(* CODESYS project filling_station_1.ecp

Project tree, tasks and I/O mapping:
  GenericDummyMasterDevice : Generic Master, WAGO, order no. None, version 1.0.0.0
  PFC200_CS_2ETH_RS : 750-8202 PFC200 2ETH RS, WAGO, order no. 0750-8202, version 1.4.1.22
    application Application
      libraries: 
      task PLC_Task (cyclic, interval t#10ms, priority 14) calls PLC_PRG
      program PLC_PRG [ST]
    DeviceAdapter
    Kbus : Kbus, WAGO, version 1.3.0.0
        unmapped channels: K-BUS diagnostics
      _4_AI_0_10V_DC_s_e : 0750-0459, WAGO, order no. 0750-0459, version 0.0.0.11
          settings: K-BUS Module slot index = 2
          unmapped channels: _IW 1, _IW 2, _IW 3, _IW 4
        DeviceAdapter
      _2_AI_4_20mA_Diff_Measurement_Input : 0750-0492, WAGO, order no. 0750-0492, version 0.0.0.7
          settings: K-BUS Module slot index = 3
          unmapped channels: _IW 1, _IW 2
        DeviceAdapter
      _8_DO_Generic : 075x-8DO, WAGO, order no. 075x-8DO, version 0.0.0.11
          settings: K-BUS Module slot index = 1
          output output1 : BOOL  // _OUT._OUT
          output output2 : BOOL  // _OUT._OUT
          unmapped channels: _OUT
        DeviceAdapter
    MODBUS
      MODBUS : MODBUS, WAGO, order no. n/a, version 1.1.1.13
    Serial
      COM1 : COM1, WAGO, version 0.0.0.19
  Library Information/
    function GetLibVersion [ST]
    function GetLibVersionNumber [ST]
    function IsLibReleased [ST]
  Project Information/
    function GetTextProperty [ST]
    function GetTextProperty2 [ST]
    function GetNumberProperty [ST]
    function GetBooleanProperty [ST]
    function GetVersionProperty [ST]
    function GetCompany [ST]
    function GetTitle [ST]
    function GetVersion [ST]
*)

// PFC200_CS_2ETH_RS/Application/PLC_PRG
PROGRAM PLC_PRG
VAR
	Controller_OP_reversed: INT;
	vrValvePosition: INT;
	Water_Valve_Open: BOOL;
	Water_Valve_Close: BOOL;
	set: INT;
END_VAR

output1:=TRUE;
output2:=TRUE;

END_PROGRAM

// Library Information/GetLibVersion
// This function has been automatically generated from the project information.
FUNCTION GetLibVersion : VERSION
VAR_INPUT
	
END_VAR

GetLibVersion.uiMajor := 0;
GetLibVersion.uiMinor := 0;
GetLibVersion.uiServicePack := 0;
GetLibVersion.uiPatch := 0;

END_FUNCTION

// Library Information/GetLibVersionNumber
// This function has been automatically generated from the project information.
FUNCTION GetLibVersionNumber : DWORD
VAR_INPUT
	
END_VAR

GetLibVersionNumber := 0;

END_FUNCTION

// Library Information/IsLibReleased
// This function has been automatically generated from the project information.
FUNCTION IsLibReleased : BOOL
VAR_INPUT
	
END_VAR

IsLibReleased := FALSE;

END_FUNCTION

// Project Information/GetTextProperty
// This function has been automatically generated from the project information.
{attribute 'signature_flag' := '1073741824'}
{attribute 'register_in_runtime'}
FUNCTION GetTextProperty : WSTRING
VAR_INPUT
	stKey: WSTRING;
END_VAR

IF stKey = "Project" THEN
	GetTextProperty := "filling_station_1";
ELSE
	GetTextProperty := "";
END_IF

END_FUNCTION

// Project Information/GetTextProperty2
// This function has been automatically generated from the project information.
{attribute 'signature_flag' := '1073741824'}
{attribute 'register_in_runtime'}
FUNCTION GetTextProperty2 : POINTER TO WSTRING
VAR_INPUT
	stKey: WSTRING;
END_VAR

IF stKey = "Project" THEN
	GetTextProperty2 := ADR("filling_station_1");
ELSE
	GetTextProperty2 := ADR("");
END_IF

END_FUNCTION

// Project Information/GetNumberProperty
// This function has been automatically generated from the project information.
{attribute 'signature_flag' := '1073741824'}
{attribute 'register_in_runtime'}
FUNCTION GetNumberProperty : DINT
VAR_INPUT
	stKey: WSTRING;
END_VAR

GetNumberProperty := 0;

END_FUNCTION

// Project Information/GetBooleanProperty
// This function has been automatically generated from the project information.
{attribute 'signature_flag' := '1073741824'}
{attribute 'register_in_runtime'}
FUNCTION GetBooleanProperty : BOOL
VAR_INPUT
	stKey: WSTRING;
END_VAR

GetBooleanProperty := FALSE;

END_FUNCTION

// Project Information/GetVersionProperty
// This function has been automatically generated from the project information.
{attribute 'signature_flag' := '1073741824'}
{attribute 'register_in_runtime'}
FUNCTION GetVersionProperty : VERSION
VAR_INPUT
	stKey: WSTRING;
END_VAR

	GetVersionProperty.uiMajor := 0;
	GetVersionProperty.uiMinor := 0;
	GetVersionProperty.uiServicePack := 0;
	GetVersionProperty.uiPatch := 0;

END_FUNCTION

// Project Information/GetCompany
// This function has been automatically generated from the project information.
{attribute 'signature_flag' := '1073741824'}
{attribute 'register_in_runtime'}
FUNCTION GetCompany : WSTRING
VAR_INPUT
	
END_VAR

GetCompany := "";

END_FUNCTION

// Project Information/GetTitle
// This function has been automatically generated from the project information.
{attribute 'signature_flag' := '1073741824'}
{attribute 'register_in_runtime'}
FUNCTION GetTitle : WSTRING
VAR_INPUT
	
END_VAR

GetTitle := "";

END_FUNCTION

// Project Information/GetVersion
// This function has been automatically generated from the project information.
{attribute 'signature_flag' := '1073741824'}
{attribute 'register_in_runtime'}
FUNCTION GetVersion : VERSION
VAR_INPUT
	
END_VAR

GetVersion.uiMajor := 0;
GetVersion.uiMinor := 0;
GetVersion.uiServicePack := 0;
GetVersion.uiPatch := 0;

END_FUNCTION
